Fanuc KAREL source: kc00036.KL

-- PROVISIONAL review KL for V940-1; original PC SHA256 f77e933cd163b64f337197e5e9583c7c8ac59482584466f4c0cc51d07052e9c9
-- Incomplete behavior may be omitted. Consult companion uncertainty JSON. Do not deploy.
PROGRAM KC00036
%NOLOCKGROUP
BEGIN
  -- V9_ZERO_TABLE_METADATA_HINT layout=0002_ascii; no indexed target words; source/name/runtime held
  -- UNRESOLVED_PC offsets 5-15; opcodes 27,31,23
  -- UNRESOLVED_PC offsets 20-24; opcodes 7F
END KC00036
